ABB RAPID module: Module1Practica2.mod

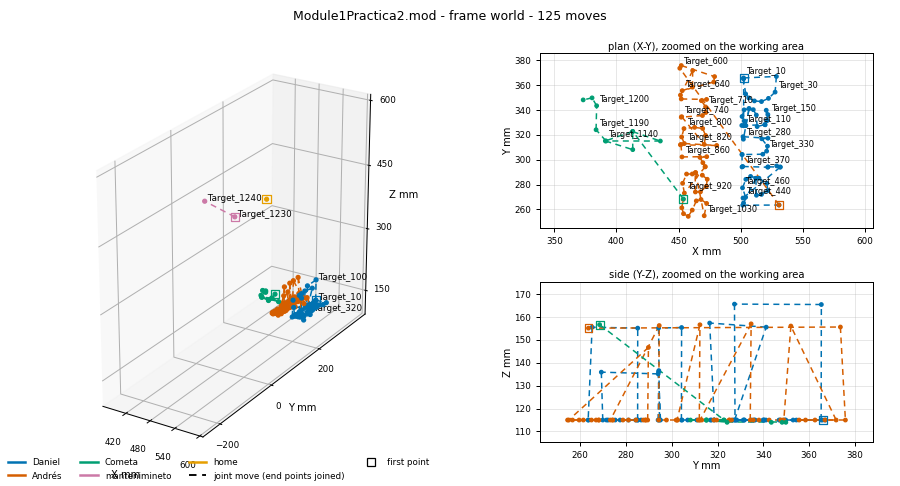
[picture p0: tool path of Module1Practica2.mod in frame world, 125 of 125 moves have a stored position in this frame; points joined in program order, loops and branches not executed]
MODULE Module1
        PERS tooldata Marcador:=[TRUE,[[103.94,0,160.94],[0.923879533,0,0.382683432,0]],[1,[0,0,1],[1,0,0,0],0,0,0]];
    TASK PERS wobjdata Workobject_1:=[FALSE,TRUE,"",[[541.896841495,226.498734393,114],[0,-0.00456097,0.999989599,0]],[[0,0,0],[1,0,0,0]]];
    CONST robtarget Target_10:=[[38.319,139.751,-1],[1,0,0,0],[0,0,0,0],[9E+09,9E+09,9E+09,9E+09,9E+09,9E+09]];
    CONST robtarget Target_20:=[[11.866,140.688,-1],[1,0,0,0],[0,-1,1,0],[9E+09,9E+09,9E+09,9E+09,9E+09,9E+09]];
    CONST robtarget Target_30:=[[13.022,128.112,-1],[1,0,0,0],[0,-1,1,0],[9E+09,9E+09,9E+09,9E+09,9E+09,9E+09]];
    CONST robtarget Target_40:=[[18.387,123.12,-1],[1,0,0,0],[0,-1,1,0],[9E+09,9E+09,9E+09,9E+09,9E+09,9E+09]];
    CONST robtarget Target_50:=[[24.061,120.604,-1],[1,0,0,0],[0,-1,1,0],[9E+09,9E+09,9E+09,9E+09,9E+09,9E+09]];
    CONST robtarget Target_60:=[[29.75,121.174,-1],[1,0,0,0],[0,-1,1,0],[9E+09,9E+09,9E+09,9E+09,9E+09,9E+09]];
    CONST robtarget Target_70:=[[34.273,123.631,-1],[1,0,0,0],[0,-1,1,0],[9E+09,9E+09,9E+09,9E+09,9E+09,9E+09]];
    CONST robtarget Target_80:=[[36.75,126.872,-1],[1,0,0,0],[0,-1,1,0],[9E+09,9E+09,9E+09,9E+09,9E+09,9E+09]];
    CONST robtarget Target_90:=[[38.293,139.132,-1],[1,0,0,0],[0,-1,1,0],[9E+09,9E+09,9E+09,9E+09,9E+09,9E+09]];
    CONST robtarget Target_100:=[[38.258,139.222,-51.484],[1,0,0,0],[0,-1,1,0],[9E+09,9E+09,9E+09,9E+09,9E+09,9E+09]];
    CONST robtarget Target_110:=[[38.572,101.258,-51.667],[1,0,0,0],[0,-1,1,0],[9E+09,9E+09,9E+09,9E+09,9E+09,9E+09]];
    CONST robtarget Target_120:=[[40.059,101.504,-1],[1,0,0,0],[0,-1,1,0],[9E+09,9E+09,9E+09,9E+09,9E+09,9E+09]];
    CONST robtarget Target_130:=[[21.258,101.883,-1],[1,0,0,0],[0,-1,1,0],[9E+09,9E+09,9E+09,9E+09,9E+09,9E+09]];
    CONST robtarget Target_140:=[[19.779,105.3,-1],[1,0,0,0],[0,-1,1,0],[9E+09,9E+09,9E+09,9E+09,9E+09,9E+09]];
    CONST robtarget Target_150:=[[19.021,110.098,-1],[1,0,0,0],[0,-1,1,0],[9E+09,9E+09,9E+09,9E+09,9E+09,9E+09]];
    CONST robtarget Target_160:=[[20.294,113.58,-1],[1,0,0,0],[0,-1,1,0],[9E+09,9E+09,9E+09,9E+09,9E+09,9E+09]];
    CONST robtarget Target_170:=[[19.658,105.402,-1],[1,0,0,0],[0,-1,1,0],[9E+09,9E+09,9E+09,9E+09,9E+09,9E+09]];
    CONST robtarget Target_180:=[[21.559,102.046,-1],[1,0,0,0],[0,-1,1,0],[9E+09,9E+09,9E+09,9E+09,9E+09,9E+09]];
    CONST robtarget Target_190:=[[27.734,100.497,-1],[1,0,0,0],[0,-1,1,0],[9E+09,9E+09,9E+09,9E+09,9E+09,9E+09]];
    CONST robtarget Target_200:=[[28.286,109.755,-1],[1,0,0,0],[0,-1,1,0],[9E+09,9E+09,9E+09,9E+09,9E+09,9E+09]];
    CONST robtarget Target_210:=[[30.701,114.126,-1],[1,0,0,0],[0,0,0,0],[9E+09,9E+09,9E+09,9E+09,9E+09,9E+09]];
    CONST robtarget Target_220:=[[34.194,114.963,-1],[1,0,0,0],[0,0,0,0],[9E+09,9E+09,9E+09,9E+09,9E+09,9E+09]];
    CONST robtarget Target_230:=[[38.098,114.071,-1],[1,0,0,0],[0,0,0,0],[9E+09,9E+09,9E+09,9E+09,9E+09,9E+09]];
    CONST robtarget Target_240:=[[39.813,108.727,-1],[1,0,0,0],[0,0,0,0],[9E+09,9E+09,9E+09,9E+09,9E+09,9E+09]];
    CONST robtarget Target_250:=[[38.113,105.103,-1],[1,0,0,0],[0,0,0,0],[9E+09,9E+09,9E+09,9E+09,9E+09,9E+09]];
    CONST robtarget Target_260:=[[36.781,101.301,-1],[1,0,0,0],[0,0,0,0],[9E+09,9E+09,9E+09,9E+09,9E+09,9E+09]];
    CONST robtarget Target_270:=[[34.075,115.071,-41.592],[1,0,0,0],[0,0,0,0],[9E+09,9E+09,9E+09,9E+09,9E+09,9E+09]];
    CONST robtarget Target_280:=[[38.908,90.431,-43.386],[1,0,0,0],[0,0,0,0],[9E+09,9E+09,9E+09,9E+09,9E+09,9E+09]];
    CONST robtarget Target_290:=[[39.18,92.444,-1],[1,0,0,0],[0,0,0,0],[9E+09,9E+09,9E+09,9E+09,9E+09,9E+09]];
    CONST robtarget Target_300:=[[19.137,91.012,-1],[1,0,0,0],[0,0,0,0],[9E+09,9E+09,9E+09,9E+09,9E+09,9E+09]];
    CONST robtarget Target_310:=[[24.091,90.627,-1],[1,0,0,0],[0,0,0,0],[9E+09,9E+09,9E+09,9E+09,9E+09,9E+09]];
    CONST robtarget Target_320:=[[19.554,84.639,-1],[1,0,0,0],[0,0,0,0],[9E+09,9E+09,9E+09,9E+09,9E+09,9E+09]];
    CONST robtarget Target_330:=[[20.275,80.652,-1],[1,0,0,0],[0,0,0,0],[9E+09,9E+09,9E+09,9E+09,9E+09,9E+09]];
    CONST robtarget Target_340:=[[23.374,78.201,-1],[1,0,0,0],[0,0,0,0],[9E+09,9E+09,9E+09,9E+09,9E+09,9E+09]];
    CONST robtarget Target_350:=[[40.121,78.077,-1],[1,0,0,0],[0,-2,1,0],[9E+09,9E+09,9E+09,9E+09,9E+09,9E+09]];
    CONST robtarget Target_360:=[[40.05,78.16,-41.432],[1,0,0,0],[0,0,0,0],[9E+09,9E+09,9E+09,9E+09,9E+09,9E+09]];
    CONST robtarget Target_370:=[[40.207,68.113,-41.218],[1,0,0,0],[0,0,0,0],[9E+09,9E+09,9E+09,9E+09,9E+09,9E+09]];
    CONST robtarget Target_380:=[[39.604,68.48,-1],[1,0,0,0],[0,-2,1,0],[9E+09,9E+09,9E+09,9E+09,9E+09,9E+09]];
    CONST robtarget Target_390:=[[19.519,67.705,-1],[1,0,0,0],[0,-2,1,0],[9E+09,9E+09,9E+09,9E+09,9E+09,9E+09]];
    CONST robtarget Target_400:=[[19.281,68.017,-22.601],[1,0,0,0],[0,0,0,0],[9E+09,9E+09,9E+09,9E+09,9E+09,9E+09]];
    CONST robtarget Target_410:=[[9.379,67.823,-22.07],[1,0,0,0],[0,0,0,0],[9E+09,9E+09,9E+09,9E+09,9E+09,9E+09]];
    CONST robtarget Target_420:=[[12.265,68.663,-1],[1,0,0,0],[0,0,0,0],[9E+09,9E+09,9E+09,9E+09,9E+09,9E+09]];
    CONST robtarget Target_430:=[[9.507,67.645,-21.164],[1,0,0,0],[0,0,0,0],[9E+09,9E+09,9E+09,9E+09,9E+09,9E+09]];
    CONST robtarget Target_440:=[[39.638,43.069,-21.93],[1,0,0,0],[0,-2,1,0],[9E+09,9E+09,9E+09,9E+09,9E+09,9E+09]];
    CONST robtarget Target_450:=[[37.53,43.686,-1],[1,0,0,0],[0,-2,1,0],[9E+09,9E+09,9E+09,9E+09,9E+09,9E+09]];
    CONST robtarget Target_460:=[[39.95,51.275,-1],[1,0,0,0],[0,-2,1,0],[9E+09,9E+09,9E+09,9E+09,9E+09,9E+09]];
    CONST robtarget Target_470:=[[37.21,58.106,-1],[1,0,0,0],[0,-2,1,0],[9E+09,9E+09,9E+09,9E+09,9E+09,9E+09]];
    CONST robtarget Target_480:=[[33.378,60.419,-1],[1,0,0,0],[0,-2,1,0],[9E+09,9E+09,9E+09,9E+09,9E+09,9E+09]];
    CONST robtarget Target_490:=[[26.633,58.914,-1],[1,0,0,0],[0,-2,1,0],[9E+09,9E+09,9E+09,9E+09,9E+09,9E+09]];
    CONST robtarget Target_500:=[[20.33,54.771,-1],[1,0,0,0],[0,-2,1,0],[9E+09,9E+09,9E+09,9E+09,9E+09,9E+09]];
    CONST robtarget Target_510:=[[19.65,48.933,-1],[1,0,0,0],[0,-2,1,0],[9E+09,9E+09,9E+09,9E+09,9E+09,9E+09]];
    CONST robtarget Target_520:=[[24.731,45.879,-1],[1,0,0,0],[0,-2,1,0],[9E+09,9E+09,9E+09,9E+09,9E+09,9E+09]];
    CONST robtarget Target_530:=[[28.796,45.214,-1],[1,0,0,0],[0,-2,1,0],[9E+09,9E+09,9E+09,9E+09,9E+09,9E+09]];
    CONST robtarget Target_540:=[[29.153,58.846,-1],[1,0,0,0],[0,-2,1,0],[9E+09,9E+09,9E+09,9E+09,9E+09,9E+09]];
    CONST robtarget Target_550:=[[29.122,58.879,-41.172],[1,0,0,0],[0,0,0,0],[9E+09,9E+09,9E+09,9E+09,9E+09,9E+09]];
    CONST robtarget Target_560:=[[39.224,39.042,-41.564],[1,0,0,0],[0,0,0,0],[9E+09,9E+09,9E+09,9E+09,9E+09,9E+09]];
    CONST robtarget Target_570:=[[39.906,37.32,-1],[1,0,0,0],[0,-2,1,0],[9E+09,9E+09,9E+09,9E+09,9E+09,9E+09]];
    CONST robtarget Target_580:=[[10.718,37.174,-1],[1,0,0,0],[0,-2,1,0],[9E+09,9E+09,9E+09,9E+09,9E+09,9E+09]];
    CONST robtarget Home_10:=[[593.569,0.329,510.811],[0,0,1,0],[0,-1,0,0],[9E+09,9E+09,9E+09,9E+09,9E+09,9E+09]];
    CONST robtarget Target_590:=[[10.726,37.185,-41.149],[1,0,0,0],[0,0,0,0],[9E+09,9E+09,9E+09,9E+09,9E+09,9E+09]];
    CONST robtarget Target_600:=[[89.566,148.012,-41.651],[1,0,0,0],[0,-1,1,0],[9E+09,9E+09,9E+09,9E+09,9E+09,9E+09]];
    CONST robtarget Target_610:=[[88.346,150.188,-1],[1,0,0,0],[0,-1,1,0],[9E+09,9E+09,9E+09,9E+09,9E+09,9E+09]];
    CONST robtarget Target_620:=[[61.636,141.033,-1],[1,0,0,0],[0,-1,1,0],[9E+09,9E+09,9E+09,9E+09,9E+09,9E+09]];
    CONST robtarget Target_630:=[[62.322,136.67,-1],[1,0,0,0],[0,-1,1,0],[9E+09,9E+09,9E+09,9E+09,9E+09,9E+09]];
    CONST robtarget Target_640:=[[87.737,129.96,-1],[1,0,0,0],[0,-1,1,0],[9E+09,9E+09,9E+09,9E+09,9E+09,9E+09]];
    CONST robtarget Target_650:=[[79.488,132.683,-1],[1,0,0,0],[0,-1,1,0],[9E+09,9E+09,9E+09,9E+09,9E+09,9E+09]];
    CONST robtarget Target_660:=[[79.222,146.063,-1],[1,0,0,0],[0,-1,1,0],[9E+09,9E+09,9E+09,9E+09,9E+09,9E+09]];
    CONST robtarget Target_670:=[[89.225,126.363,-42.082],[1,0,0,0],[0,-1,1,0],[9E+09,9E+09,9E+09,9E+09,9E+09,9E+09]];
    CONST robtarget Target_680:=[[88.617,123.28,-1],[1,0,0,0],[0,-1,1,0],[9E+09,9E+09,9E+09,9E+09,9E+09,9E+09]];
    CONST robtarget Target_690:=[[68.241,122.712,-1],[1,0,0,0],[0,-1,1,0],[9E+09,9E+09,9E+09,9E+09,9E+09,9E+09]];
    CONST robtarget Target_700:=[[72.424,121.778,-1],[1,0,0,0],[0,0,0,0],[9E+09,9E+09,9E+09,9E+09,9E+09,9E+09]];
    CONST robtarget Target_710:=[[69.086,116.698,-1],[1,0,0,0],[0,0,0,0],[9E+09,9E+09,9E+09,9E+09,9E+09,9E+09]];
    CONST robtarget Target_720:=[[68.921,112.221,-1],[1,0,0,0],[0,0,0,0],[9E+09,9E+09,9E+09,9E+09,9E+09,9E+09]];
    CONST robtarget Target_730:=[[71.692,109.778,-1],[1,0,0,0],[0,0,0,0],[9E+09,9E+09,9E+09,9E+09,9E+09,9E+09]];
    CONST robtarget Target_740:=[[88.744,108.601,-1],[1,0,0,0],[0,0,0,0],[9E+09,9E+09,9E+09,9E+09,9E+09,9E+09]];
    CONST robtarget Target_750:=[[88.381,108.987,-43.033],[1,0,0,0],[0,0,0,0],[9E+09,9E+09,9E+09,9E+09,9E+09,9E+09]];
    CONST robtarget Target_760:=[[70.452,86.52,-1],[1,0,0,0],[0,-2,1,0],[9E+09,9E+09,9E+09,9E+09,9E+09,9E+09]];
    CONST robtarget Target_770:=[[69.304,93.713,-1],[1,0,0,0],[0,-2,1,0],[9E+09,9E+09,9E+09,9E+09,9E+09,9E+09]];
    CONST robtarget Target_780:=[[71.589,99.363,-1],[1,0,0,0],[0,-2,1,0],[9E+09,9E+09,9E+09,9E+09,9E+09,9E+09]];
    CONST robtarget Target_790:=[[78.052,100.332,-1],[1,0,0,0],[0,-2,1,0],[9E+09,9E+09,9E+09,9E+09,9E+09,9E+09]];
    CONST robtarget Target_800:=[[86.644,99.405,-1],[1,0,0,0],[0,-2,1,0],[9E+09,9E+09,9E+09,9E+09,9E+09,9E+09]];
    CONST robtarget Target_810:=[[88.561,92.677,-1],[1,0,0,0],[0,-2,1,0],[9E+09,9E+09,9E+09,9E+09,9E+09,9E+09]];
    CONST robtarget Target_820:=[[86.49,87.397,-1],[1,0,0,0],[0,-2,1,0],[9E+09,9E+09,9E+09,9E+09,9E+09,9E+09]];
    CONST robtarget Target_830:=[[60.424,85.578,-1],[1,0,0,0],[0,-2,1,0],[9E+09,9E+09,9E+09,9E+09,9E+09,9E+09]];
    CONST robtarget Target_840:=[[89.606,86.354,-1],[1,0,0,0],[0,-2,1,0],[9E+09,9E+09,9E+09,9E+09,9E+09,9E+09]];
    CONST robtarget Target_850:=[[89.218,86.623,-42.633],[1,0,0,0],[0,0,0,0],[9E+09,9E+09,9E+09,9E+09,9E+09,9E+09]];
    CONST robtarget Target_860:=[[88.453,76.624,-1],[1,0,0,0],[0,-2,1,0],[9E+09,9E+09,9E+09,9E+09,9E+09,9E+09]];
    CONST robtarget Target_870:=[[68.552,76.649,-1],[1,0,0,0],[0,-2,1,0],[9E+09,9E+09,9E+09,9E+09,9E+09,9E+09]];
    CONST robtarget Target_880:=[[73.968,76.096,-1],[1,0,0,0],[0,-2,1,0],[9E+09,9E+09,9E+09,9E+09,9E+09,9E+09]];
    CONST robtarget Target_890:=[[71.681,71.821,-1],[1,0,0,0],[0,-2,1,0],[9E+09,9E+09,9E+09,9E+09,9E+09,9E+09]];
    CONST robtarget Target_900:=[[69.962,68.407,-1],[1,0,0,0],[0,-2,1,0],[9E+09,9E+09,9E+09,9E+09,9E+09,9E+09]];
    CONST robtarget Target_910:=[[69.772,68.658,-42.29],[1,0,0,0],[0,0,0,0],[9E+09,9E+09,9E+09,9E+09,9E+09,9E+09]];
    CONST robtarget Target_920:=[[86.8,47.443,-1],[1,0,0,0],[0,-2,1,0],[9E+09,9E+09,9E+09,9E+09,9E+09,9E+09]];
    CONST robtarget Target_930:=[[88.139,55.376,-1],[1,0,0,0],[0,-2,1,0],[9E+09,9E+09,9E+09,9E+09,9E+09,9E+09]];
    CONST robtarget Target_940:=[[84.892,62.817,-1],[1,0,0,0],[0,-2,1,0],[9E+09,9E+09,9E+09,9E+09,9E+09,9E+09]];
    CONST robtarget Target_950:=[[80.319,62.803,-1],[1,0,0,0],[0,-2,1,0],[9E+09,9E+09,9E+09,9E+09,9E+09,9E+09]];
    CONST robtarget Target_960:=[[72.198,61.751,-1],[1,0,0,0],[0,-2,1,0],[9E+09,9E+09,9E+09,9E+09,9E+09,9E+09]];
    CONST robtarget Target_970:=[[68.277,58.456,-1],[1,0,0,0],[0,-2,1,0],[9E+09,9E+09,9E+09,9E+09,9E+09,9E+09]];
    CONST robtarget Target_980:=[[69.072,52.793,-1],[1,0,0,0],[0,-2,1,0],[9E+09,9E+09,9E+09,9E+09,9E+09,9E+09]];
    CONST robtarget Target_990:=[[73.845,48.372,-1],[1,0,0,0],[0,-2,1,0],[9E+09,9E+09,9E+09,9E+09,9E+09,9E+09]];
    CONST robtarget Target_1000:=[[77.919,48.318,-1],[1,0,0,0],[0,-2,1,0],[9E+09,9E+09,9E+09,9E+09,9E+09,9E+09]];
    CONST robtarget Target_1010:=[[77.923,63.686,-1],[1,0,0,0],[0,-2,1,0],[9E+09,9E+09,9E+09,9E+09,9E+09,9E+09]];
    CONST robtarget Target_1020:=[[77.571,64.001,-32.73],[1,0,0,0],[0,0,0,0],[9E+09,9E+09,9E+09,9E+09,9E+09,9E+09]];
    CONST robtarget Target_1030:=[[70.991,29.117,-1],[1,0,0,0],[0,-2,1,0],[9E+09,9E+09,9E+09,9E+09,9E+09,9E+09]];
    CONST robtarget Target_1040:=[[68.964,39.024,-1],[1,0,0,0],[0,-2,1,0],[9E+09,9E+09,9E+09,9E+09,9E+09,9E+09]];
    CONST robtarget Target_1050:=[[73.446,42.217,-1],[1,0,0,0],[0,-2,1,0],[9E+09,9E+09,9E+09,9E+09,9E+09,9E+09]];
    CONST robtarget Target_1060:=[[77.253,41.124,-1],[1,0,0,0],[0,-2,1,0],[9E+09,9E+09,9E+09,9E+09,9E+09,9E+09]];
    CONST robtarget Target_1070:=[[80.575,33.745,-1],[1,0,0,0],[0,-2,1,0],[9E+09,9E+09,9E+09,9E+09,9E+09,9E+09]];
    CONST robtarget Target_1080:=[[83.837,28.738,-1],[1,0,0,0],[0,-2,1,0],[9E+09,9E+09,9E+09,9E+09,9E+09,9E+09]];
    CONST robtarget Target_1090:=[[87.636,30.913,-1],[1,0,0,0],[0,-2,1,0],[9E+09,9E+09,9E+09,9E+09,9E+09,9E+09]];
    CONST robtarget Target_1100:=[[88.957,35.665,-1],[1,0,0,0],[0,-2,1,0],[9E+09,9E+09,9E+09,9E+09,9E+09,9E+09]];
    CONST robtarget Target_1110:=[[87.818,42.435,-1],[1,0,0,0],[0,-2,1,0],[9E+09,9E+09,9E+09,9E+09,9E+09,9E+09]];
    CONST robtarget Target_1120:=[[87.597,42.763,-42.679],[1,0,0,0],[0,0,0,0],[9E+09,9E+09,9E+09,9E+09,9E+09,9E+09]];
    CONST robtarget Target_1130:=[[127.915,97.554,-1],[1,0,0,0],[0,-2,1,0],[9E+09,9E+09,9E+09,9E+09,9E+09,9E+09]];
    CONST robtarget Target_1140:=[[150.01,90.022,-1],[1,0,0,0],[0,-2,1,0],[9E+09,9E+09,9E+09,9E+09,9E+09,9E+09]];
    CONST robtarget Target_1150:=[[128.026,82.833,-1],[1,0,0,0],[0,-2,1,0],[9E+09,9E+09,9E+09,9E+09,9E+09,9E+09]];
    CONST robtarget Target_1160:=[[127.946,97.346,-1],[1,0,0,0],[0,-2,1,0],[9E+09,9E+09,9E+09,9E+09,9E+09,9E+09]];
    CONST robtarget Target_1170:=[[105.755,89.564,-1],[1,0,0,0],[0,-2,1,0],[9E+09,9E+09,9E+09,9E+09,9E+09,9E+09]];
    CONST robtarget Target_1180:=[[149.488,90.009,-1],[1,0,0,0],[0,-2,1,0],[9E+09,9E+09,9E+09,9E+09,9E+09,9E+09]];
    CONST robtarget Target_1190:=[[157.399,99.113,0],[1,0,0,0],[0,-2,1,0],[9E+09,9E+09,9E+09,9E+09,9E+09,9E+09]];
    CONST robtarget Target_1200:=[[156.762,118.436,0],[1,0,0,0],[0,-2,1,0],[9E+09,9E+09,9E+09,9E+09,9E+09,9E+09]];
    CONST robtarget Target_1210:=[[160.399,124.815,0],[1,0,0,0],[0,-1,1,0],[9E+09,9E+09,9E+09,9E+09,9E+09,9E+09]];
    CONST robtarget Target_1220:=[[167.548,123.244,0],[1,0,0,0],[0,-1,1,0],[9E+09,9E+09,9E+09,9E+09,9E+09,9E+09]];
    CONST robtarget Mantenimiento_10:=[[628.673,-0.205,987.508],[0,0,1,0],[0,0,0,0],[9E+09,9E+09,9E+09,9E+09,9E+09,9E+09]];
    CONST robtarget Target_1230:=[[595.506,-123.828,517.619],[0,0,1,0],[-1,0,-1,0],[9E+09,9E+09,9E+09,9E+09,9E+09,9E+09]];
    CONST robtarget Target_1240:=[[597.135,-235.281,591.266],[0,0,1,0],[-1,0,-1,0],[9E+09,9E+09,9E+09,9E+09,9E+09,9E+09]];
!***********************************************************
    !
    ! M?dulo:  Module1
    !
    ! Descripción:
    !   <Introduzca la descripción aquí>
    !
    ! Autor: Daniel Segura
    !
    ! Versión: 1.0
    !
    !***********************************************************


    !***********************************************************
    !
    ! Procedimiento Main
    !
    !   Este es el punto de entrada de su programa
    !
    !***********************************************************
    PROC main()
        WHILE TRUE DO
            IF DI_01=1 AND DI_02=0 THEN
                SetDO DO_01,1;
                SetDO DO_03,0;
                home;
                Daniel;
                home;
                WaitTime 15;
            ENDIF
            IF DI_02=1 AND DI_01=0 THEN
                SetDO DO_01,0;
                SetDO DO_03,1;
                mantenimineto;
                WaitTime 15;
            ENDIF
        ENDWHILE
    ENDPROC
    PROC Daniel()
        MoveJ Target_10,v400,z5,Marcador\WObj:=Workobject_1;
        MoveJ Target_20,v400,z5,Marcador\WObj:=Workobject_1;
        MoveJ Target_30,v400,z5,Marcador\WObj:=Workobject_1;
        MoveJ Target_40,v400,z5,Marcador\WObj:=Workobject_1;
        MoveJ Target_50,v400,z5,Marcador\WObj:=Workobject_1;
        MoveJ Target_60,v400,z5,Marcador\WObj:=Workobject_1;
        MoveJ Target_70,v400,z5,Marcador\WObj:=Workobject_1;
        MoveJ Target_80,v400,z5,Marcador\WObj:=Workobject_1;
        MoveJ Target_90,v400,z5,Marcador\WObj:=Workobject_1;
        MoveJ Target_100,v400,z5,Marcador\WObj:=Workobject_1;
        MoveJ Target_110,v400,z5,Marcador\WObj:=Workobject_1;
        MoveJ Target_120,v400,z5,Marcador\WObj:=Workobject_1;
        MoveJ Target_130,v400,z5,Marcador\WObj:=Workobject_1;
        MoveJ Target_140,v400,z5,Marcador\WObj:=Workobject_1;
        MoveJ Target_150,v400,z5,Marcador\WObj:=Workobject_1;
        MoveJ Target_160,v400,z5,Marcador\WObj:=Workobject_1;
        MoveJ Target_170,v400,z5,Marcador\WObj:=Workobject_1;
        MoveJ Target_180,v400,z5,Marcador\WObj:=Workobject_1;
        MoveJ Target_190,v400,z5,Marcador\WObj:=Workobject_1;
        MoveJ Target_200,v400,z5,Marcador\WObj:=Workobject_1;
        MoveJ Target_210,v400,z5,Marcador\WObj:=Workobject_1;
        MoveJ Target_220,v400,z5,Marcador\WObj:=Workobject_1;
        MoveJ Target_230,v400,z5,Marcador\WObj:=Workobject_1;
        MoveJ Target_240,v400,z5,Marcador\WObj:=Workobject_1;
        MoveJ Target_250,v400,z5,Marcador\WObj:=Workobject_1;
        MoveJ Target_260,v400,z5,Marcador\WObj:=Workobject_1;
        MoveJ Target_270,v400,z5,Marcador\WObj:=Workobject_1;
        MoveJ Target_280,v400,z5,Marcador\WObj:=Workobject_1;
        MoveJ Target_290,v400,z5,Marcador\WObj:=Workobject_1;
        MoveJ Target_300,v400,z5,Marcador\WObj:=Workobject_1;
        MoveJ Target_310,v400,z5,Marcador\WObj:=Workobject_1;
        MoveJ Target_320,v400,z5,Marcador\WObj:=Workobject_1;
        MoveJ Target_330,v400,z5,Marcador\WObj:=Workobject_1;
        MoveJ Target_340,v400,z5,Marcador\WObj:=Workobject_1;
        MoveJ Target_350,v400,z5,Marcador\WObj:=Workobject_1;
        MoveJ Target_360,v400,z5,Marcador\WObj:=Workobject_1;
        MoveJ Target_370,v400,z5,Marcador\WObj:=Workobject_1;
        MoveJ Target_380,v400,z5,Marcador\WObj:=Workobject_1;
        MoveJ Target_390,v400,z5,Marcador\WObj:=Workobject_1;
        MoveJ Target_400,v400,z5,Marcador\WObj:=Workobject_1;
        MoveJ Target_410,v400,z5,Marcador\WObj:=Workobject_1;
        MoveJ Target_420,v400,z5,Marcador\WObj:=Workobject_1;
        MoveJ Target_430,v400,z5,Marcador\WObj:=Workobject_1;
        MoveJ Target_440,v400,z5,Marcador\WObj:=Workobject_1;
        MoveJ Target_450,v400,z5,Marcador\WObj:=Workobject_1;
        MoveJ Target_460,v400,z5,Marcador\WObj:=Workobject_1;
        MoveJ Target_470,v400,z5,Marcador\WObj:=Workobject_1;
        MoveJ Target_480,v400,z5,Marcador\WObj:=Workobject_1;
        MoveJ Target_490,v400,z5,Marcador\WObj:=Workobject_1;
        MoveJ Target_500,v400,z5,Marcador\WObj:=Workobject_1;
        MoveJ Target_510,v400,z5,Marcador\WObj:=Workobject_1;
        MoveJ Target_520,v400,z5,Marcador\WObj:=Workobject_1;
        MoveJ Target_530,v400,z5,Marcador\WObj:=Workobject_1;
        MoveJ Target_540,v400,z5,Marcador\WObj:=Workobject_1;
        MoveJ Target_550,v400,z5,Marcador\WObj:=Workobject_1;
        MoveJ Target_560,v400,z5,Marcador\WObj:=Workobject_1;
        MoveJ Target_570,v400,z5,Marcador\WObj:=Workobject_1;
        MoveJ Target_580,v400,z5,Marcador\WObj:=Workobject_1;
        Andrés;
    ENDPROC
    PROC Andrés()
        MoveJ Target_590,v400,z5,Marcador\WObj:=Workobject_1;
        MoveJ Target_600,v400,z5,Marcador\WObj:=Workobject_1;
        MoveJ Target_610,v400,z5,Marcador\WObj:=Workobject_1;
        MoveJ Target_620,v400,z5,Marcador\WObj:=Workobject_1;
        MoveJ Target_630,v400,z5,Marcador\WObj:=Workobject_1;
        MoveJ Target_640,v400,z5,Marcador\WObj:=Workobject_1;
        MoveJ Target_650,v400,z5,Marcador\WObj:=Workobject_1;
        MoveJ Target_660,v400,z5,Marcador\WObj:=Workobject_1;
        MoveJ Target_670,v400,z5,Marcador\WObj:=Workobject_1;
        MoveJ Target_680,v400,z5,Marcador\WObj:=Workobject_1;
        MoveJ Target_690,v400,z5,Marcador\WObj:=Workobject_1;
        MoveJ Target_700,v400,z5,Marcador\WObj:=Workobject_1;
        MoveJ Target_710,v400,z5,Marcador\WObj:=Workobject_1;
        MoveJ Target_720,v400,z5,Marcador\WObj:=Workobject_1;
        MoveJ Target_730,v400,z5,Marcador\WObj:=Workobject_1;
        MoveJ Target_740,v400,z5,Marcador\WObj:=Workobject_1;
        MoveJ Target_750,v400,z5,Marcador\WObj:=Workobject_1;
        MoveJ Target_760,v400,z5,Marcador\WObj:=Workobject_1;
        MoveJ Target_770,v400,z5,Marcador\WObj:=Workobject_1;
        MoveJ Target_780,v400,z5,Marcador\WObj:=Workobject_1;
        MoveJ Target_790,v400,z5,Marcador\WObj:=Workobject_1;
        MoveJ Target_800,v400,z5,Marcador\WObj:=Workobject_1;
        MoveJ Target_810,v400,z5,Marcador\WObj:=Workobject_1;
        MoveJ Target_820,v400,z5,Marcador\WObj:=Workobject_1;
        MoveJ Target_830,v400,z5,Marcador\WObj:=Workobject_1;
        MoveJ Target_840,v400,z5,Marcador\WObj:=Workobject_1;
        MoveJ Target_850,v400,z5,Marcador\WObj:=Workobject_1;
        MoveJ Target_860,v400,z5,Marcador\WObj:=Workobject_1;
        MoveJ Target_870,v400,z5,Marcador\WObj:=Workobject_1;
        MoveJ Target_880,v400,z5,Marcador\WObj:=Workobject_1;
        MoveJ Target_890,v400,z5,Marcador\WObj:=Workobject_1;
        MoveJ Target_900,v400,z5,Marcador\WObj:=Workobject_1;
        MoveJ Target_910,v400,z5,Marcador\WObj:=Workobject_1;
        MoveJ Target_920,v400,z5,Marcador\WObj:=Workobject_1;
        MoveJ Target_930,v400,z5,Marcador\WObj:=Workobject_1;
        MoveJ Target_940,v400,z5,Marcador\WObj:=Workobject_1;
        MoveJ Target_950,v400,z5,Marcador\WObj:=Workobject_1;
        MoveJ Target_960,v400,z5,Marcador\WObj:=Workobject_1;
        MoveJ Target_970,v400,z5,Marcador\WObj:=Workobject_1;
        MoveJ Target_980,v400,z5,Marcador\WObj:=Workobject_1;
        MoveJ Target_990,v400,z5,Marcador\WObj:=Workobject_1;
        MoveJ Target_1000,v400,z5,Marcador\WObj:=Workobject_1;
        MoveJ Target_1010,v400,z5,Marcador\WObj:=Workobject_1;
        MoveJ Target_1020,v400,z5,Marcador\WObj:=Workobject_1;
        MoveJ Target_1030,v400,z5,Marcador\WObj:=Workobject_1;
        MoveJ Target_1040,v400,z5,Marcador\WObj:=Workobject_1;
        MoveJ Target_1050,v400,z5,Marcador\WObj:=Workobject_1;
        MoveJ Target_1060,v400,z5,Marcador\WObj:=Workobject_1;
        MoveJ Target_1070,v400,z5,Marcador\WObj:=Workobject_1;
        MoveJ Target_1080,v400,z5,Marcador\WObj:=Workobject_1;
        MoveJ Target_1090,v400,z5,Marcador\WObj:=Workobject_1;
        MoveJ Target_1100,v400,z5,Marcador\WObj:=Workobject_1;
        MoveJ Target_1110,v400,z5,Marcador\WObj:=Workobject_1;
        Cometa;
    ENDPROC
    PROC Cometa()
        MoveJ Target_1120,v400,z5,Marcador\WObj:=Workobject_1;
        MoveJ Target_1130,v400,z5,Marcador\WObj:=Workobject_1;
        MoveJ Target_1140,v400,z5,Marcador\WObj:=Workobject_1;
        MoveJ Target_1150,v400,z5,Marcador\WObj:=Workobject_1;
        MoveJ Target_1160,v400,z5,Marcador\WObj:=Workobject_1;
        MoveJ Target_1170,v400,z5,Marcador\WObj:=Workobject_1;
        MoveJ Target_1180,v400,z5,Marcador\WObj:=Workobject_1;
        MoveJ Target_1190,v400,z5,Marcador\WObj:=Workobject_1;
        MoveJ Target_1200,v400,z5,Marcador\WObj:=Workobject_1;
        MoveJ Target_1210,v400,z5,Marcador\WObj:=Workobject_1;
        MoveJ Target_1220,v400,z5,Marcador\WObj:=Workobject_1;
    ENDPROC
    PROC mantenimineto()
        MoveJ Target_1230,v100,z5,Marcador\WObj:=wobj0;
        MoveJ Target_1240,v100,z5,Marcador\WObj:=wobj0;
    ENDPROC
    PROC home()
        MoveJ Home_10,v400,z5,Marcador\WObj:=wobj0;
    ENDPROC
ENDMODULE
